// Writes a double field value, without a tag, to the stream.
FUNCTION F_WriteDouble : HRESULT
VAR_IN_OUT
    stCtx   : ST_WriteContext;
END_VAR
VAR_INPUT CONSTANT
    fValue : LREAL;
END_VAR
VAR CONSTANT
    cLength : UDINT := SIZEOF(fValue);
END_VAR
VAR
    fTmp : LREAL;
END_VAR

{warning 'TODO: Check for endianess?'}
fTmp := fValue;

F_WriteDouble := F_WriteToBuffer(stCtx, F_ToAnyType(fTmp), cLength);

END_FUNCTION

(* stored: Version 1.1.0.1
   POU F_WriteDouble: Id {bd6826a6-616d-4379-89c3-33633543bf20}, SpecialFunc None *)
